// TIA Portal project "ACT350DIN_PNET_S2B_ST13_v02 Light_V14" (V14)

(* hardware
DEVICE "S7-1200 station_1"  S7-1200 Station
   slot 0: "Rack_0"  Rack  V1.0
   slot 1: "PLC_1"  CPU 1212C AC/DC/Rly  6ES7 212-1BE40-0XB0  V4.1
DEVICE "GSD device_1"  GSD.Device.PN
   slot 0: "Rack"  Rail  V1.0
   slot 0: "ACT350"  MT-ACT30XXXXXX  V2.6.1
*)

// ===== PLC "PLC_1"  CPU 1212C AC/DC/Rly =====

VAR_GLOBAL   // PLC tag table "Default tag table"
   "rMBCommandValue" AT %QD256 : Real;
   "wMBChannelMask" AT %QW260 : Word;
   "wMBCommand" AT %QW262 : Word;
   "bOutput0" AT %Q0.0 : Bool;
   "bAlarm" AT %I261.4 : Bool;
   "bCenterZero" AT %I261.5 : Bool;
   "BMBDeviceStatus_Upper" AT %IB260 : Byte;
   "wMBResponse" AT %IW262 : Word;
   "intSequenceNumber" AT %MW270 : Int;
   "rWeightData" AT %ID256 : DWord;
   "BMBDeviceStatus_Lower" AT %IB261 : Byte;
   "BDeviceStatus_Upper" AT %MB3 : Byte;
   "BDeviceStatus_Lower" AT %MB2 : Byte;
   "WDeviceStatus_Word" AT %MW2 : Word;
   "bSequenceNumber_bit0" AT %M271.0 : Bool;
   "bSequenceNumber_bit1" AT %M271.1 : Bool;
   "bHeartBeat_FAILED" AT %M1.7 : Bool;
   "DI01" AT %I0.0 : Bool;
   "DI04" AT %I0.3 : Bool;
   "DI02" AT %I0.1 : Bool;
   "DI03" AT %I0.2 : Bool;
END_VAR

TYPE "Measuring Block Read"
VERSION : 0.1
   STRUCT
      Element_1 : Struct
         "FP Data" : Real;
         "Measuring Status Read" : "MB Measuring Status Bits";
         "Command Response Word" : Word;
      END_STRUCT;
   END_STRUCT;
END_TYPE

TYPE "MB Measuring Status Bits"
VERSION : 0.1
   STRUCT
      Element_1 : Struct
         "Sequence Bit 0" : Bool;
         "Sequence Bit 1" : Bool;
         "Heart Bit" : Bool;
         "Data OK" : Bool;
         Alarm : Bool;
         "Center of Zero" : Bool;
         "In Motion" : Bool;
         "Net Mode" : Bool;
         "Alternate Weight unit" : Bool;
         "Device Specific Bit 1" : Bool;
         "Device Specific Bit 2" : Bool;
         "Device Specific Bit 3" : Bool;
         "Device Specific Bit 4" : Bool;
         "Device Specific Bit 5" : Bool;
         "Device Specific Bit 6" : Bool;
         "Device Specific Bit 7" : Bool;
      END_STRUCT;
   END_STRUCT;
END_TYPE

DATA_BLOCK "Cyclic Input Data"   // DB3
{ S7_Optimized_Access := 'FALSE' }
VERSION : 0.1
   VAR
      Static_1 : "Measuring Block Read";
   END_VAR
BEGIN
END_DATA_BLOCK

DATA_BLOCK "Cyclic Command"   // DB17
{ S7_Optimized_Access := 'TRUE' }
VERSION : 0.1
   VAR
      ByteOrderTest_Cyclic : Bool;   // Cyclic command to perform Byte Order Test
      ReportDefault_Cyclic : Bool;   // Cyclic command to request default weight data from device
      PresetTare_Cyclic : Bool;   // Cyclic command to perform preset tare onto device
      ReportGross_Cyclic : Bool;   // Cyclic command to request gross weight data from device
      ReportTare_Cyclic : Bool;   // Cyclic command to request tare weight data from device
      ReportNet_Cyclic : Bool;   // Cyclic command to request net weight data from device
      TareStable_Cyclic : Bool;   // Cyclic command to perform tare when stable onto device
      ZeroStable_Cyclic : Bool;   // Cyclic command to perform zero when stable onto device
      ClearTare_Cyclic : Bool;   // Cyclic command to perform clear tare onto device
      Noop_Cyclic : Bool;   // Cyclic command to perform no-operation
      WriteComparator1_Cyclic : Bool;   // Cyclic command to write comparator 1 value onto device
      Comparator1_Value : Real;   // Comparator 1 value to be written onto device
      PreTare_Weight : Real;   // Pre-tare weight value to be written onto device
      Always_ON : Bool;   // internal bit used for programming
      CommandHistory : Word;   // Cyclic command which has been executed earlier
      CommandExecuted : Bool;   // Bit to show that new cyclic command has been aknowledged and executed by device
      SequenceNumberMemory : Int;   // Sequence number increment by 1 from 0 to 3 everytime a new command has been executed
      ByteOrder_OK : Bool;
   END_VAR
BEGIN
END_DATA_BLOCK

// folder: System blocks/Program resources

DATA_BLOCK "CommandAck_TON"   // DB1
{ S7_Optimized_Access := 'TRUE' }
AUTHOR : Simatic
FAMILY : IEC
NAME : IEC_TMR
VERSION : 1.0
// stored: InstanceOfName IEC_TIMER
"IEC_TIMER"
BEGIN
END_DATA_BLOCK

DATA_BLOCK "ByteOrder_TON"   // DB6
{ S7_Optimized_Access := 'TRUE' }
AUTHOR : Simatic
FAMILY : IEC
NAME : IEC_TMR
VERSION : 1.0
// stored: InstanceOfName IEC_TIMER
"IEC_TIMER"
BEGIN
END_DATA_BLOCK

DATA_BLOCK "HeartBeat_TIMER"   // DB13
{ S7_Optimized_Access := 'TRUE' }
AUTHOR : Simatic
FAMILY : IEC
NAME : IEC_TMR
VERSION : 1.0
// stored: InstanceOfName IEC_TIMER
"IEC_TIMER"
BEGIN
END_DATA_BLOCK

// folder: (top level)

ORGANIZATION_BLOCK "CyclicProgram"   // OB200, LAD, ProgramCycle
TITLE = Cyclic Commands Program
{ S7_Optimized_Access := 'TRUE' }
VERSION : 0.1
   VAR_INPUT
      Initial_Call : Bool;   // Initial call of this OB
      Remanence : Bool;   // =True, if remanent data are available
   END_VAR
   VAR_TEMP
      bTemp1 : Bool;
      bTemp2 : Bool;
      bTemp3 : Bool;
      bTemp4 : Bool;
      bTemp5 : Bool;
      bTemp6 : Bool;
      bTemp7 : Bool;
      bTemp8 : Bool;
      bTemp9 : Bool;
      bUpdateDisplay1 : Bool;
      bUpdateDisplay2 : Bool;
      bTareLatch : Bool;
      bClearTareLatch : Bool;
      bResetHearBeatTimer : Bool;
   END_VAR
   VAR_TEMP   // added for the SCL form of the ladder/FBD networks
      _w1 : Bool;
      _w2 : Bool;
      _w3 : Bool;
      _w4 : Bool;
      _w5 : Bool;
      _w6 : Bool;
      _w7 : Bool;
      _w8 : Bool;
      _w9 : Bool;
      _w10 : Bool;
      _w11 : Bool;
   END_VAR
BEGIN

REGION Network 1: Read in all cyclical input data
   // PLC reads in 1st block of cyclical data (measuring block) from SAI device. Measuring Block (MB) input consists of 4 words. 
   // MB Measuring Value = 2 words = 32-bit floating point single precision weight data;
   // MB Device Status = 1 word =  SAI device status (e.g. Heartbeat, Data OK, Alarm, Net Mode, Center of Zero, sequence bits etc.)
   // MB Response = 1 word = SAI device response to new cyclic commands
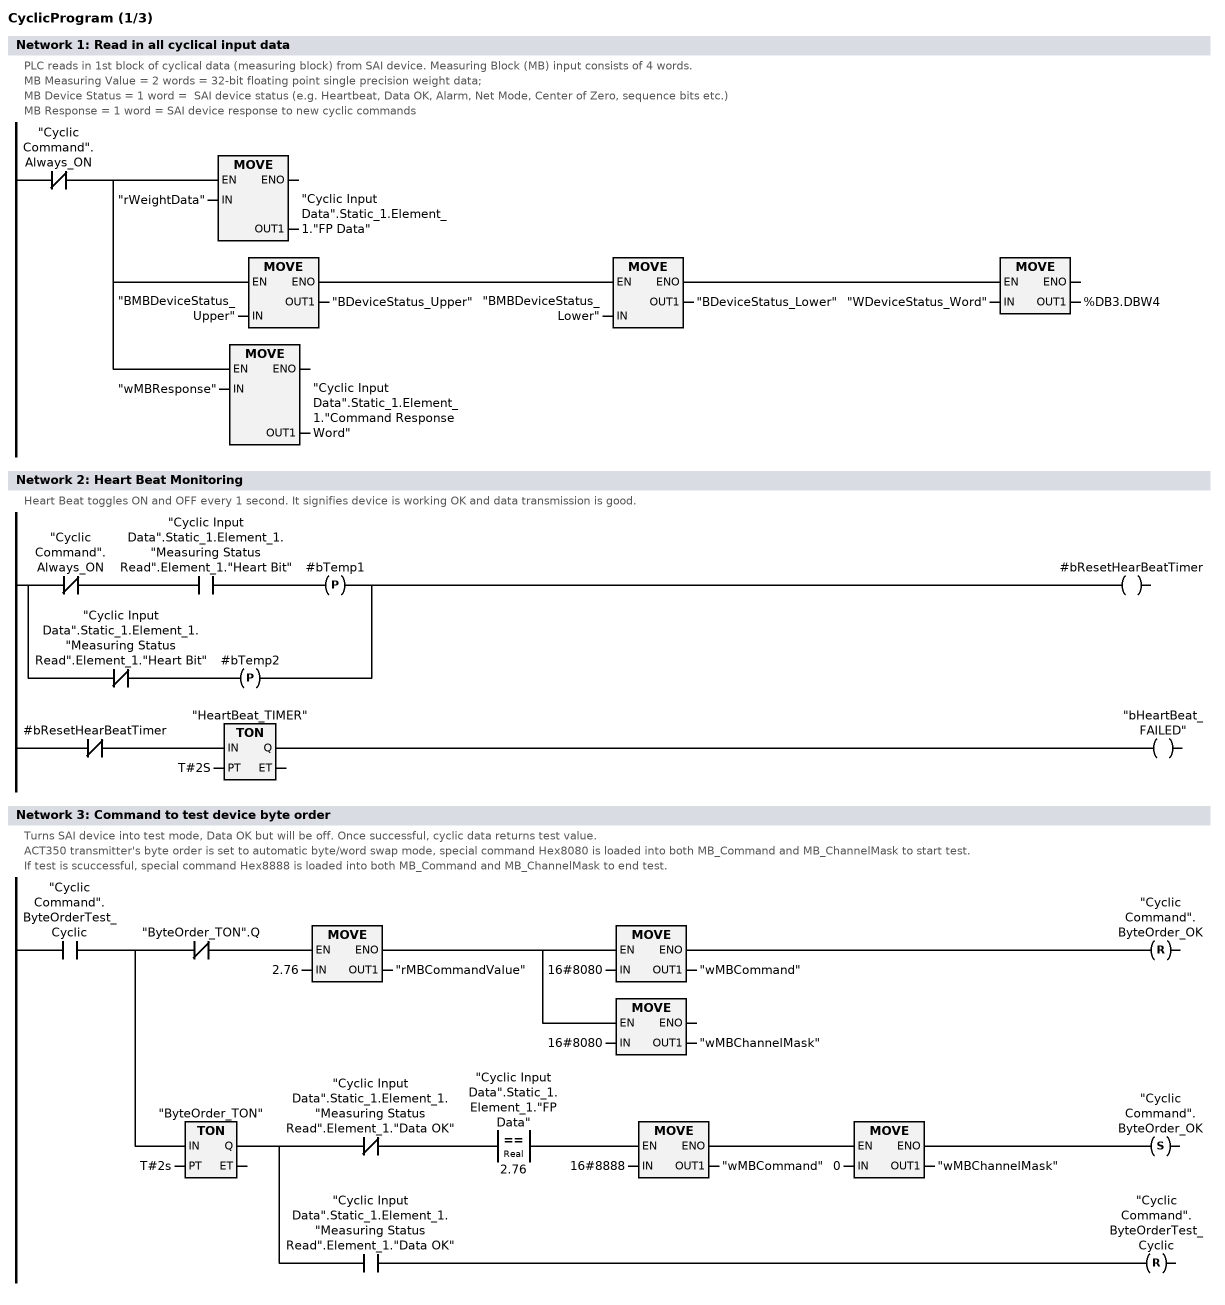
   RUNG wire#powerrail
      I_Contact( "Cyclic Command".Always_ON )
      wire#w1
      Move(in := "rWeightData", out1 => "Cyclic Input Data".Static_1.Element_1."FP Data")
   END_RUNG
   RUNG wire#w1
      Move(in := "BMBDeviceStatus_Upper", out1 => "BDeviceStatus_Upper")
      Move(in := "BMBDeviceStatus_Lower", out1 => "BDeviceStatus_Lower")
      Move(in := "WDeviceStatus_Word", out1 => %DB3.DBW4)
   END_RUNG
   RUNG wire#w1
      Move(in := "wMBResponse", out1 => "Cyclic Input Data".Static_1.Element_1."Command Response Word")
   END_RUNG
   // the same network as SCL:
   IF NOT "Cyclic Command".Always_ON THEN
       "Cyclic Input Data".Static_1.Element_1."FP Data" := "rWeightData";
       "BDeviceStatus_Upper" := "BMBDeviceStatus_Upper";
       "BDeviceStatus_Lower" := "BMBDeviceStatus_Lower";
       %DB3.DBW4 := "WDeviceStatus_Word";
       "Cyclic Input Data".Static_1.Element_1."Command Response Word" := "wMBResponse";
   END_IF;
END_REGION

REGION Network 2: Heart Beat Monitoring
   // Heart Beat toggles ON and OFF every 1 second. It signifies device is working OK and data transmission is good.
   #_w1 := NOT "Cyclic Command".Always_ON AND "Cyclic Input Data".Static_1.Element_1."Measuring Status Read".Element_1."Heart Bit";
   #_w2 := #_w1 AND NOT #bTemp1;   // rising edge
   #bTemp1 := #_w1;
   #_w3 := NOT "Cyclic Input Data".Static_1.Element_1."Measuring Status Read".Element_1."Heart Bit" AND NOT #bTemp2;   // rising edge
   #bTemp2 := NOT "Cyclic Input Data".Static_1.Element_1."Measuring Status Read".Element_1."Heart Bit";
   #bResetHearBeatTimer := #_w2 OR #_w3;
   "HeartBeat_TIMER".TON(IN := NOT #bResetHearBeatTimer, PT := T#2S);
   "bHeartBeat_FAILED" := "HeartBeat_TIMER".Q;
END_REGION

REGION Network 3: Command to test device byte order
   // Turns SAI device into test mode, Data OK but will be off. Once successful, cyclic data returns test value. 
   // ACT350 transmitter's byte order is set to automatic byte/word swap mode, special command Hex8080 is loaded into both MB_Command and MB_ChannelMask to start test.
   // If test is scuccessful, special command Hex8888 is loaded into both MB_Command and MB_ChannelMask to end test.
   IF "Cyclic Command".ByteOrderTest_Cyclic AND NOT "ByteOrder_TON".Q THEN
       "rMBCommandValue" := 2.76;
       "wMBCommand" := 16#8080;
       "Cyclic Command".ByteOrder_OK := FALSE;
       "wMBChannelMask" := 16#8080;
   END_IF;
   "ByteOrder_TON".TON(IN := "Cyclic Command".ByteOrderTest_Cyclic, PT := T#2s);
   IF "ByteOrder_TON".Q AND NOT "Cyclic Input Data".Static_1.Element_1."Measuring Status Read".Element_1."Data OK" AND ("Cyclic Input Data".Static_1.Element_1."FP Data" = 2.76) THEN
       "wMBCommand" := 16#8888;
       "wMBChannelMask" := 0;
       "Cyclic Command".ByteOrder_OK := TRUE;
   END_IF;
   IF "ByteOrder_TON".Q AND "Cyclic Input Data".Static_1.Element_1."Measuring Status Read".Element_1."Data OK" THEN
       "Cyclic Command".ByteOrderTest_Cyclic := FALSE;
   END_IF;
END_REGION

REGION Network 4: List of Cyclic Commands
   // Command 0 - Report Default Weight Value
   // Command 1 - Report Gross Weight Value
   // Command 2 - Report Tare Weight Value
   // Command 3 - Report Net Weight Value
   // Command 400 - Tare When Stable
   // Command 401 - Zero When Stable
   // Command 402 - Clear Tare
   // Command 403 - Tare Immediate
   // Command 404 - Zero Immediate
   // Command 201 - Preset Tare (by giving a preset tare weight)
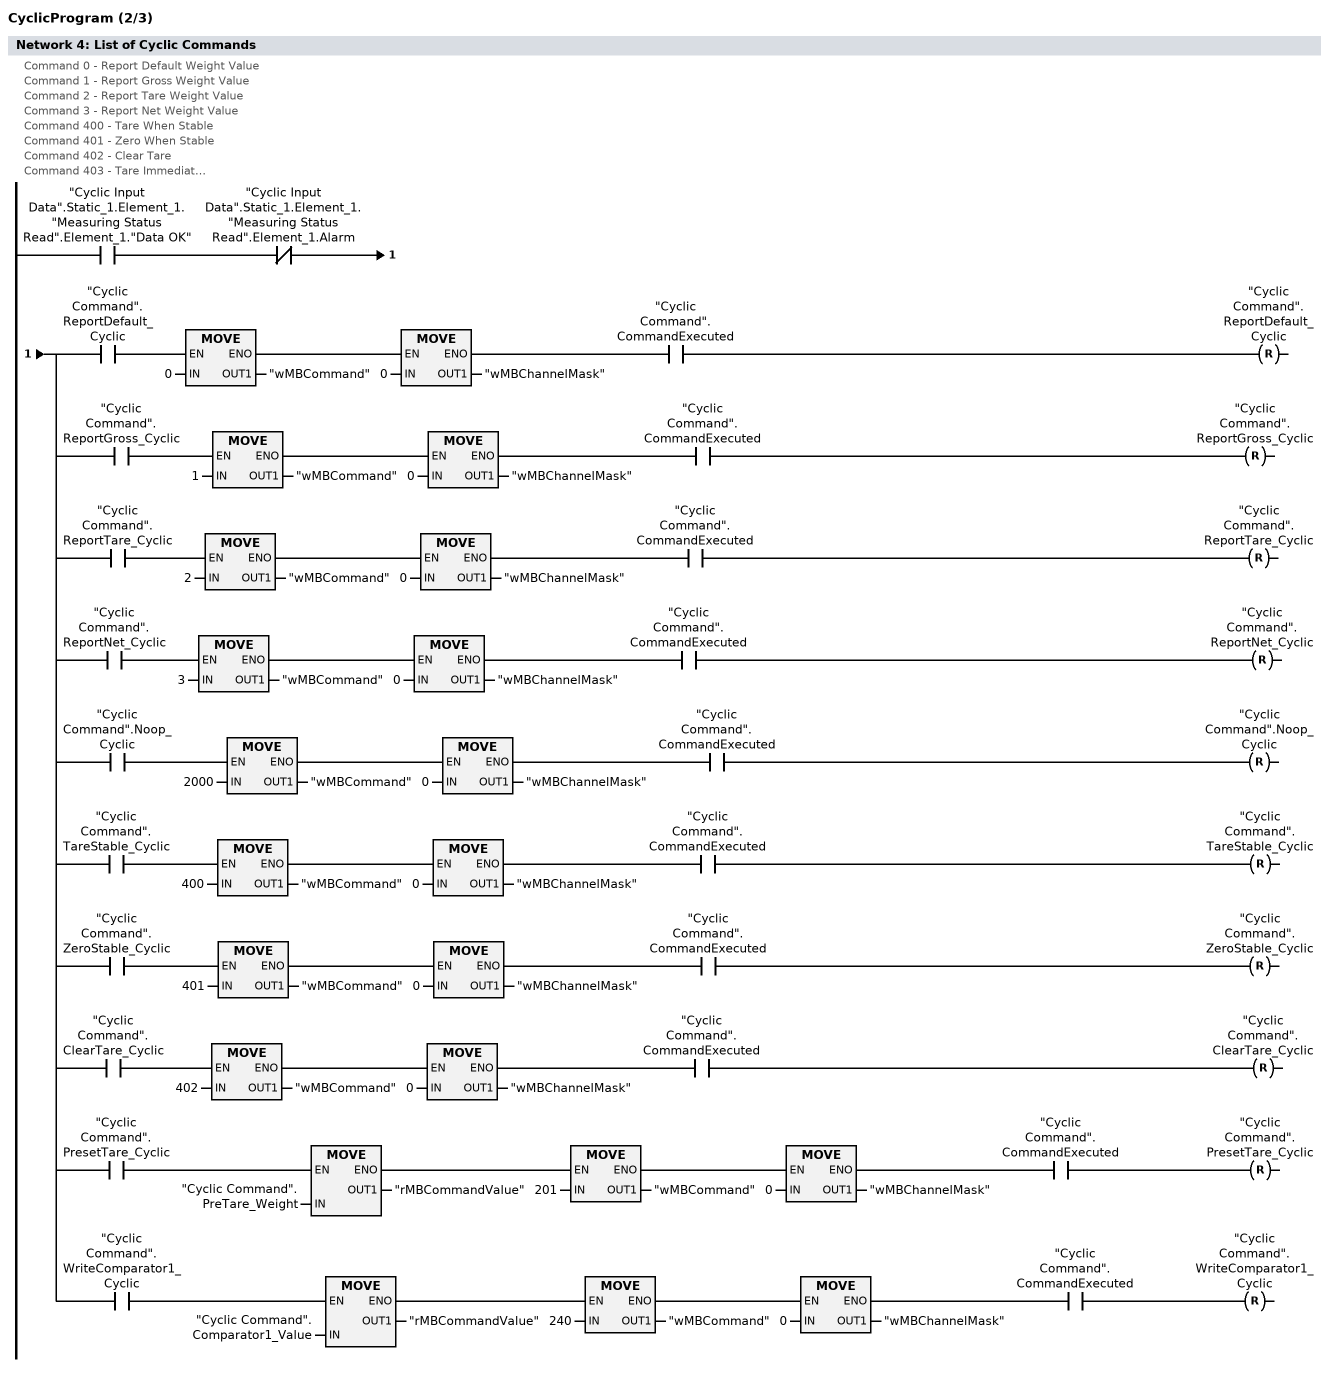
   RUNG wire#powerrail
      Contact( "Cyclic Input Data".Static_1.Element_1."Measuring Status Read".Element_1."Data OK" )
      I_Contact( "Cyclic Input Data".Static_1.Element_1."Measuring Status Read".Element_1.Alarm )
      wire#w1
      Contact( "Cyclic Command".ReportDefault_Cyclic )
      Move(in := 0, out1 => "wMBCommand")
      Move(in := 0, out1 => "wMBChannelMask")
      Contact( "Cyclic Command".CommandExecuted )
      R_Coil( "Cyclic Command".ReportDefault_Cyclic )
   END_RUNG
   RUNG wire#w1
      Contact( "Cyclic Command".ReportGross_Cyclic )
      Move(in := 1, out1 => "wMBCommand")
      Move(in := 0, out1 => "wMBChannelMask")
      Contact( "Cyclic Command".CommandExecuted )
      R_Coil( "Cyclic Command".ReportGross_Cyclic )
   END_RUNG
   RUNG wire#w1
      Contact( "Cyclic Command".ReportTare_Cyclic )
      Move(in := 2, out1 => "wMBCommand")
      Move(in := 0, out1 => "wMBChannelMask")
      Contact( "Cyclic Command".CommandExecuted )
      R_Coil( "Cyclic Command".ReportTare_Cyclic )
   END_RUNG
   RUNG wire#w1
      Contact( "Cyclic Command".ReportNet_Cyclic )
      Move(in := 3, out1 => "wMBCommand")
      Move(in := 0, out1 => "wMBChannelMask")
      Contact( "Cyclic Command".CommandExecuted )
      R_Coil( "Cyclic Command".ReportNet_Cyclic )
   END_RUNG
   RUNG wire#w1
      Contact( "Cyclic Command".Noop_Cyclic )
      Move(in := 2000, out1 => "wMBCommand")
      Move(in := 0, out1 => "wMBChannelMask")
      Contact( "Cyclic Command".CommandExecuted )
      R_Coil( "Cyclic Command".Noop_Cyclic )
   END_RUNG
   RUNG wire#w1
      Contact( "Cyclic Command".TareStable_Cyclic )
      Move(in := 400, out1 => "wMBCommand")
      Move(in := 0, out1 => "wMBChannelMask")
      Contact( "Cyclic Command".CommandExecuted )
      R_Coil( "Cyclic Command".TareStable_Cyclic )
   END_RUNG
   RUNG wire#w1
      Contact( "Cyclic Command".ZeroStable_Cyclic )
      Move(in := 401, out1 => "wMBCommand")
      Move(in := 0, out1 => "wMBChannelMask")
      Contact( "Cyclic Command".CommandExecuted )
      R_Coil( "Cyclic Command".ZeroStable_Cyclic )
   END_RUNG
   RUNG wire#w1
      Contact( "Cyclic Command".ClearTare_Cyclic )
      Move(in := 402, out1 => "wMBCommand")
      Move(in := 0, out1 => "wMBChannelMask")
      Contact( "Cyclic Command".CommandExecuted )
      R_Coil( "Cyclic Command".ClearTare_Cyclic )
   END_RUNG
   RUNG wire#w1
      Contact( "Cyclic Command".PresetTare_Cyclic )
      Move(in := "Cyclic Command".PreTare_Weight, out1 => "rMBCommandValue")
      Move(in := 201, out1 => "wMBCommand")
      Move(in := 0, out1 => "wMBChannelMask")
      Contact( "Cyclic Command".CommandExecuted )
      R_Coil( "Cyclic Command".PresetTare_Cyclic )
   END_RUNG
   RUNG wire#w1
      Contact( "Cyclic Command".WriteComparator1_Cyclic )
      Move(in := "Cyclic Command".Comparator1_Value, out1 => "rMBCommandValue")
      Move(in := 240, out1 => "wMBCommand")
      Move(in := 0, out1 => "wMBChannelMask")
      Contact( "Cyclic Command".CommandExecuted )
      R_Coil( "Cyclic Command".WriteComparator1_Cyclic )
   END_RUNG
   // the same network as SCL:
   #_w1 := "Cyclic Input Data".Static_1.Element_1."Measuring Status Read".Element_1."Data OK" AND NOT "Cyclic Input Data".Static_1.Element_1."Measuring Status Read".Element_1.Alarm;
   #_w2 := #_w1 AND "Cyclic Command".ReportDefault_Cyclic;
   IF #_w2 THEN
       "wMBCommand" := 0;
       "wMBChannelMask" := 0;
   END_IF;
   IF #_w2 AND "Cyclic Command".CommandExecuted THEN "Cyclic Command".ReportDefault_Cyclic := FALSE; END_IF;
   #_w3 := #_w1 AND "Cyclic Command".ReportGross_Cyclic;
   IF #_w3 THEN
       "wMBCommand" := 1;
       "wMBChannelMask" := 0;
   END_IF;
   IF #_w3 AND "Cyclic Command".CommandExecuted THEN "Cyclic Command".ReportGross_Cyclic := FALSE; END_IF;
   #_w4 := #_w1 AND "Cyclic Command".ReportTare_Cyclic;
   IF #_w4 THEN
       "wMBCommand" := 2;
       "wMBChannelMask" := 0;
   END_IF;
   IF #_w4 AND "Cyclic Command".CommandExecuted THEN "Cyclic Command".ReportTare_Cyclic := FALSE; END_IF;
   #_w5 := #_w1 AND "Cyclic Command".ReportNet_Cyclic;
   IF #_w5 THEN
       "wMBCommand" := 3;
       "wMBChannelMask" := 0;
   END_IF;
   IF #_w5 AND "Cyclic Command".CommandExecuted THEN "Cyclic Command".ReportNet_Cyclic := FALSE; END_IF;
   #_w6 := #_w1 AND "Cyclic Command".Noop_Cyclic;
   IF #_w6 THEN
       "wMBCommand" := 2000;
       "wMBChannelMask" := 0;
   END_IF;
   IF #_w6 AND "Cyclic Command".CommandExecuted THEN "Cyclic Command".Noop_Cyclic := FALSE; END_IF;
   #_w7 := #_w1 AND "Cyclic Command".TareStable_Cyclic;
   IF #_w7 THEN
       "wMBCommand" := 400;
       "wMBChannelMask" := 0;
   END_IF;
   IF #_w7 AND "Cyclic Command".CommandExecuted THEN "Cyclic Command".TareStable_Cyclic := FALSE; END_IF;
   #_w8 := #_w1 AND "Cyclic Command".ZeroStable_Cyclic;
   IF #_w8 THEN
       "wMBCommand" := 401;
       "wMBChannelMask" := 0;
   END_IF;
   IF #_w8 AND "Cyclic Command".CommandExecuted THEN "Cyclic Command".ZeroStable_Cyclic := FALSE; END_IF;
   #_w9 := #_w1 AND "Cyclic Command".ClearTare_Cyclic;
   IF #_w9 THEN
       "wMBCommand" := 402;
       "wMBChannelMask" := 0;
   END_IF;
   IF #_w9 AND "Cyclic Command".CommandExecuted THEN "Cyclic Command".ClearTare_Cyclic := FALSE; END_IF;
   #_w10 := #_w1 AND "Cyclic Command".PresetTare_Cyclic;
   IF #_w10 THEN
       "rMBCommandValue" := "Cyclic Command".PreTare_Weight;
       "wMBCommand" := 201;
       "wMBChannelMask" := 0;
   END_IF;
   IF #_w10 AND "Cyclic Command".CommandExecuted THEN "Cyclic Command".PresetTare_Cyclic := FALSE; END_IF;
   #_w11 := #_w1 AND "Cyclic Command".WriteComparator1_Cyclic;
   IF #_w11 THEN
       "rMBCommandValue" := "Cyclic Command".Comparator1_Value;
       "wMBCommand" := 240;
       "wMBChannelMask" := 0;
   END_IF;
   IF #_w11 AND "Cyclic Command".CommandExecuted THEN
       "Cyclic Command".WriteComparator1_Cyclic := FALSE;
   END_IF;
END_REGION

REGION Network 5: Command acknowledgement from Device for every new PLC command
   // Here the programming checks whether a new cyclic command has been issued and wait for acknowledgement.
   // Upon successfull execution of any cyclic command, SAI device will copy the command value from MB Command into MB Response word. 
   // Then lastly device will increment the sequence bits.
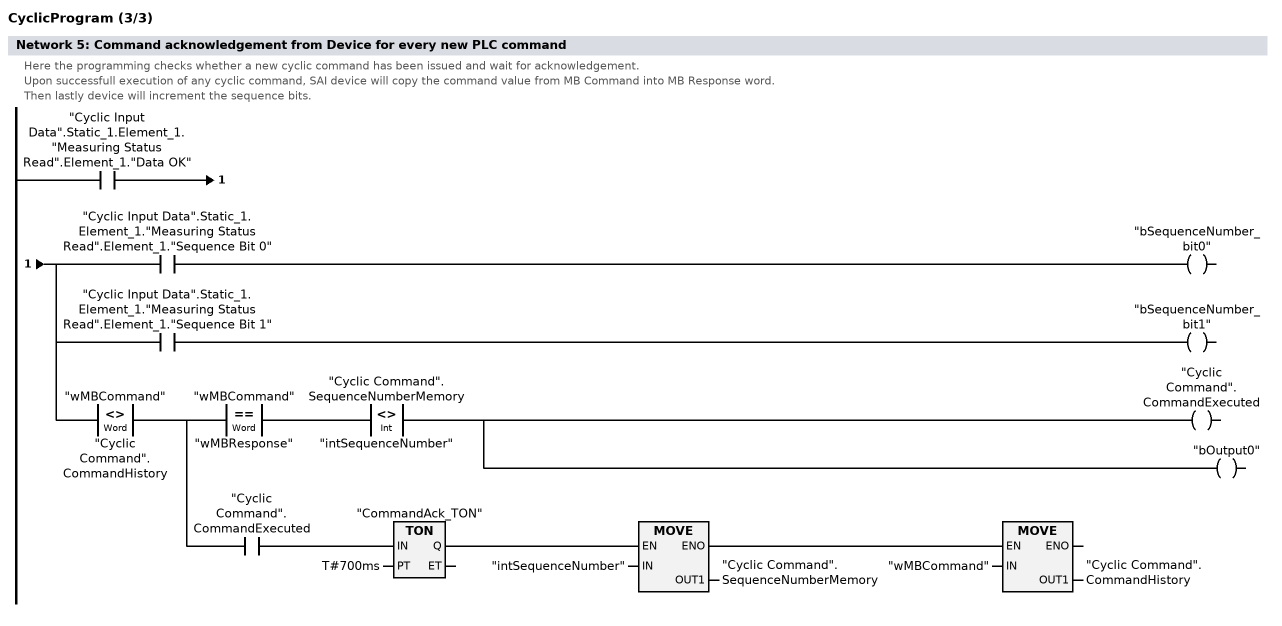
   "bSequenceNumber_bit0" := "Cyclic Input Data".Static_1.Element_1."Measuring Status Read".Element_1."Data OK" AND "Cyclic Input Data".Static_1.Element_1."Measuring Status Read".Element_1."Sequence Bit 0";
   "bSequenceNumber_bit1" := "Cyclic Input Data".Static_1.Element_1."Measuring Status Read".Element_1."Data OK" AND "Cyclic Input Data".Static_1.Element_1."Measuring Status Read".Element_1."Sequence Bit 1";
   #_w1 := "Cyclic Input Data".Static_1.Element_1."Measuring Status Read".Element_1."Data OK" AND ("wMBCommand" <> "Cyclic Command".CommandHistory);
   "Cyclic Command".CommandExecuted := #_w1 AND ("wMBCommand" = "wMBResponse") AND ("Cyclic Command".SequenceNumberMemory <> "intSequenceNumber");
   "bOutput0" := "Cyclic Command".CommandExecuted;
   "CommandAck_TON".TON(IN := #_w1 AND "Cyclic Command".CommandExecuted, PT := T#700ms);
   IF "CommandAck_TON".Q THEN
       "Cyclic Command".SequenceNumberMemory := "intSequenceNumber";
       "Cyclic Command".CommandHistory := "wMBCommand";
   END_IF;
END_REGION
END_ORGANIZATION_BLOCK